FUNCTION_BLOCK changeEventM262_2 (* Basic Function Block Type *)
  (* Standard: 61499-2 *)
  (* Version 0.0, 5/23/2025, azam_w, Schneider Electric, Template *)
  PACKAGE Main;
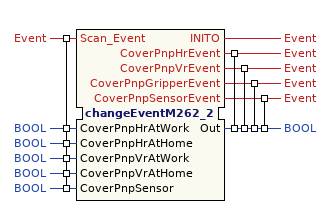
  EVENT_INPUT
    Scan_Event WITH CoverPnpHrAtWork, CoverPnpHrAtHome, CoverPnpVrAtWork, CoverPnpVrAtHome, CoverPnpSensor;
  END_EVENT
  EVENT_OUTPUT
    INITO; (* Initialization Confirm *)
    CoverPnpHrEvent WITH Out;
    CoverPnpVrEvent WITH Out;
    CoverPnpGripperEvent WITH Out;
    CoverPnpSensorEvent WITH Out;
  END_EVENT
  VAR_INPUT
    CoverPnpHrAtWork : BOOL;
    CoverPnpHrAtHome : BOOL;
    CoverPnpVrAtWork : BOOL;
    CoverPnpVrAtHome : BOOL;
    CoverPnpSensor : BOOL;
  END_VAR
  VAR_OUTPUT
    Out : BOOL;
  END_VAR
  VAR
    CoverPnpHrAtWork_PrevVal : BOOL;
    CoverPnpHrAtHome_PrevVal : BOOL;
    CoverPnpVrAtWork_PrevVal : BOOL;
    CoverPnpVrAtHome_PrevVal : BOOL;
    CoverPnpGripperClosed_PrevVal : BOOL;
    CoverPnpGripperOpened_PrevVal : BOOL;
    CoverPnpSensor_PreVal : BOOL;
  END_VAR
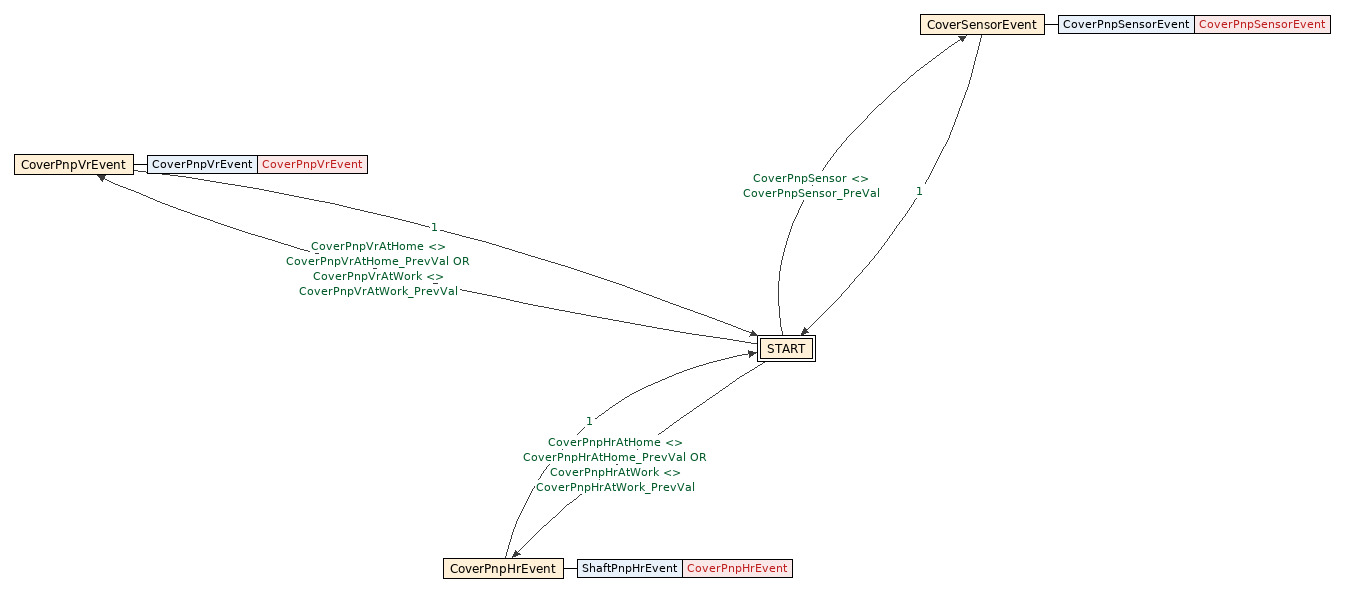
  EC_STATES
    START; (* Initial State *)
    CoverPnpHrEvent : ShaftPnpHrEvent -> CoverPnpHrEvent;
    CoverPnpVrEvent : CoverPnpVrEvent -> CoverPnpVrEvent;
    CoverSensorEvent : CoverPnpSensorEvent -> CoverPnpSensorEvent;
  END_STATES
  EC_TRANSITIONS
    START TO CoverPnpHrEvent := CoverPnpHrAtHome <> CoverPnpHrAtHome_PrevVal OR CoverPnpHrAtWork <> CoverPnpHrAtWork_PrevVal;
    CoverPnpHrEvent TO START := 1;
    START TO CoverPnpVrEvent := CoverPnpVrAtHome <> CoverPnpVrAtHome_PrevVal OR CoverPnpVrAtWork <> CoverPnpVrAtWork_PrevVal;
    CoverPnpVrEvent TO START := 1;
    START TO CoverSensorEvent := CoverPnpSensor <> CoverPnpSensor_PreVal;
    CoverSensorEvent TO START := 1;
  END_TRANSITIONS
  ALGORITHM INIT IN ST: (* Initialization algorithm *)
;
  END_ALGORITHM
  ALGORITHM ShaftPnpHrEvent IN ST:
;
IF CoverPnpHrAtHome <> CoverPnpHrAtHome_PrevVal THEN
	CoverPnpHrAtHome_PrevVal := CoverPnpHrAtHome;
	Out := CoverPnpHrAtHome;
END_IF;

IF CoverPnpHrAtWork <> CoverPnpHrAtWork_PrevVal THEN
	CoverPnpHrAtWork_PrevVal := CoverPnpHrAtWork;
	Out := CoverPnpHrAtWork;
END_IF;
  END_ALGORITHM
  ALGORITHM CoverPnpSensorEvent IN ST:
;
IF CoverPnpSensor <> CoverPnpSensor_PreVal THEN
	CoverPnpSensor_PreVal := CoverPnpSensor;
	Out := CoverPnpSensor;
END_IF;
  END_ALGORITHM
  ALGORITHM CoverPnpVrEvent IN ST:
;
IF CoverPnpVrAtHome <> CoverPnpVrAtHome_PrevVal THEN
	CoverPnpVrAtHome_PrevVal := CoverPnpVrAtHome;
	Out := CoverPnpVrAtHome;
END_IF;

IF CoverPnpVrAtWork <> CoverPnpVrAtWork_PrevVal THEN
	CoverPnpVrAtWork_PrevVal := CoverPnpVrAtWork;
	Out := CoverPnpVrAtWork;
END_IF;
  END_ALGORITHM
END_FUNCTION_BLOCK
